PROGRAM HMI_Door_Toggle
VAR
	dwDoorFlag: DWORD;
	dwDoor1: DWORD;
	dwDoor2: DWORD;
	dwDoor3: DWORD;
	dwDoor4: DWORD;
	bDoorFlag : BOOL;
END_VAR

//Door Interlock Indicator Logic
	IF GV_LIFT.DOOR_1_INDICATOR_IN AND GV_LIFT.DOOR_2_INDICATOR_IN AND GV_LIFT.DOOR_3_INDICATOR_IN AND GV_LIFT.DOOR_4_INDICATOR_IN THEN
		dwDoorFlag := GV_HMI.dwGreen;
		bDoorFlag := FALSE;
	ELSE dwDoorFlag := GV_HMI.dwRed;
		bDoorFlag := TRUE;
	END_IF 
	
	//Door 1 Indicator
		IF GV_LIFT.DOOR_1_INDICATOR_OUT THEN
			dwDoor1 := GV_HMI.dwRed;
		ELSIF GV_Lift.DOOR_1_INDICATOR_LATCH_OUT THEN
			dwDoor1 := GV_HMI.dwYellow;
		ELSE dwDoor1 := GV_HMI.dwGreen;
		END_IF
	//Door 2 Indicator
		IF GV_LIFT.DOOR_2_INDICATOR_OUT THEN
			dwDoor2 := GV_HMI.dwRed;
		ELSIF GV_Lift.DOOR_2_INDICATOR_LATCH_OUT THEN
			dwDoor2 := GV_HMI.dwYellow;
		ELSE dwDoor2 := GV_HMI.dwGreen;
		END_IF
	//Door 3 Indicator
		IF GV_LIFT.DOOR_3_INDICATOR_OUT THEN
			dwDoor3 := GV_HMI.dwRed;
		ELSIF GV_Lift.DOOR_3_INDICATOR_LATCH_OUT THEN
			dwDoor3 := GV_HMI.dwYellow;
		ELSE dwDoor3 := GV_HMI.dwGreen;
		END_IF
	//Door 4 Indicator
		IF GV_LIFT.DOOR_4_INDICATOR_OUT THEN
			dwDoor4 := GV_HMI.dwRed;
		ELSIF GV_Lift.DOOR_4_INDICATOR_LATCH_OUT THEN
			dwDoor4 := GV_HMI.dwYellow;
		ELSE dwDoor4 := GV_HMI.dwGreen;
		END_IF

END_PROGRAM

(* stored: Version 1.1.0.1, ProductVersion 3.1.4022.12
   POU HMI_Door_Toggle: Id {4268ac57-f08a-4dd4-aeaa-43a224c81dac}, SpecialFunc None *)
